TYPE ST_4Bytes :
STRUCT
	Byte1	: BYTE;
	Byte2	: BYTE;
	Byte3	: BYTE;
	Byte4	: BYTE;
END_STRUCT
END_TYPE

(* stored: Version 1.1.0.1, ProductVersion 3.1.4024.12
   DUT ST_4Bytes: Id {e02c2b4c-8ecc-4bc1-92f9-75027e9eae4a} *)
